PROGRAM main
VAR
	Power_On AT %IX0.0 : bool;
	Machine_Ready AT %QX0.0 : bool;
	TON0 : TON;
END_VAR

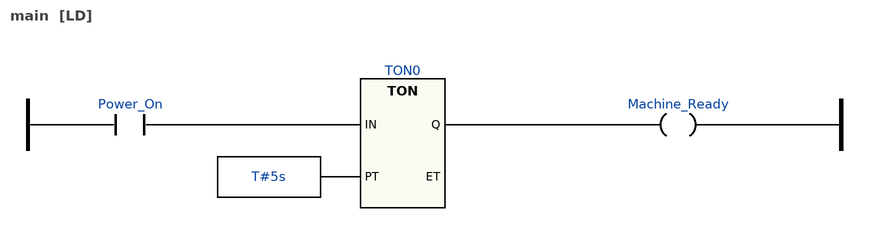
(* LD diagram, written out as Structured Text *)
TON0(IN := Power_On, PT := T#5s);
Machine_Ready := TON0.Q;
END_PROGRAM
